TYPE "UDT_Marking StringToChar"
VERSION : 0.1
   STRUCT
      "Char" : Array[0..127] of Char;
   END_STRUCT;

END_TYPE

